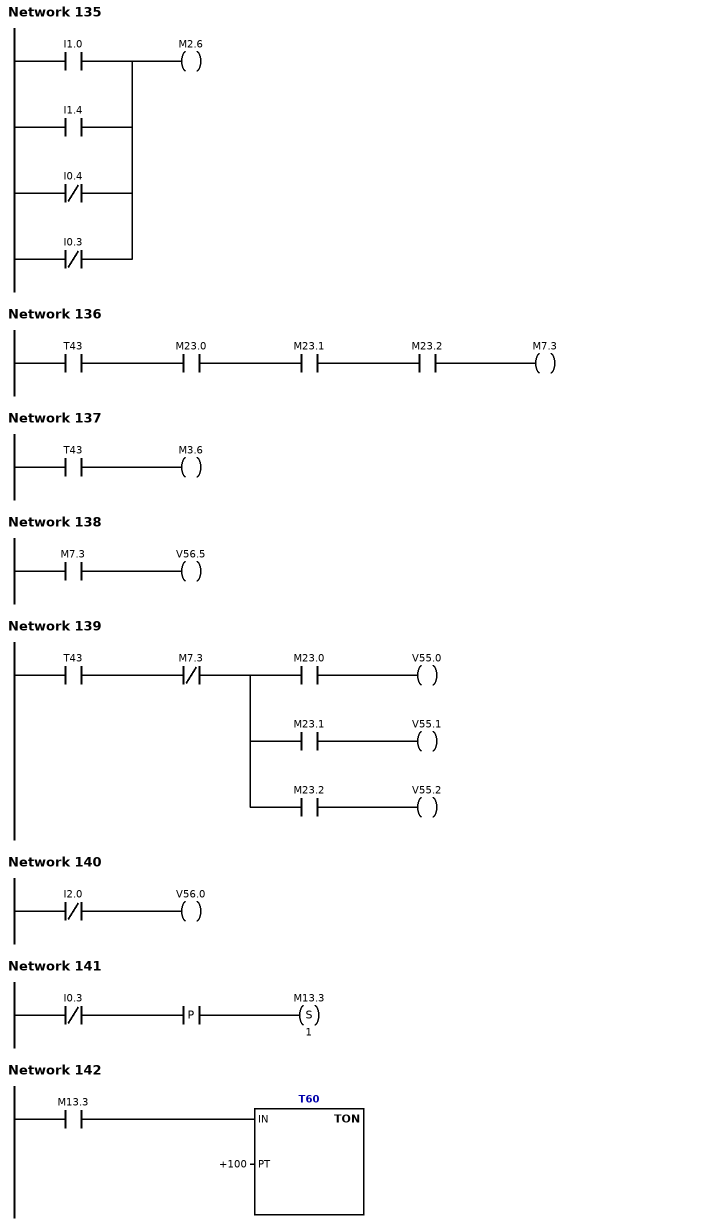
[picture p24: OB1 networks 135-142]
Network 135
LD     I1.0
O      I1.4
ON     I0.4
ON     I0.3
=      M2.6
Network 136
LD     T43
A      M23.0
A      M23.1
A      M23.2
=      M7.3
Network 137
LD     T43
=      M3.6
Network 138
LD     M7.3
=      V56.5
Network 139
LD     T43
AN     M7.3
LPS
A      M23.0
=      V55.0
LRD
A      M23.1
=      V55.1
LPP
A      M23.2
=      V55.2
Network 140
LDN    I2.0
=      V56.0
Network 141
LDN    I0.3
EU
S      M13.3, 1
Network 142
LD     M13.3
TON    T60, +100
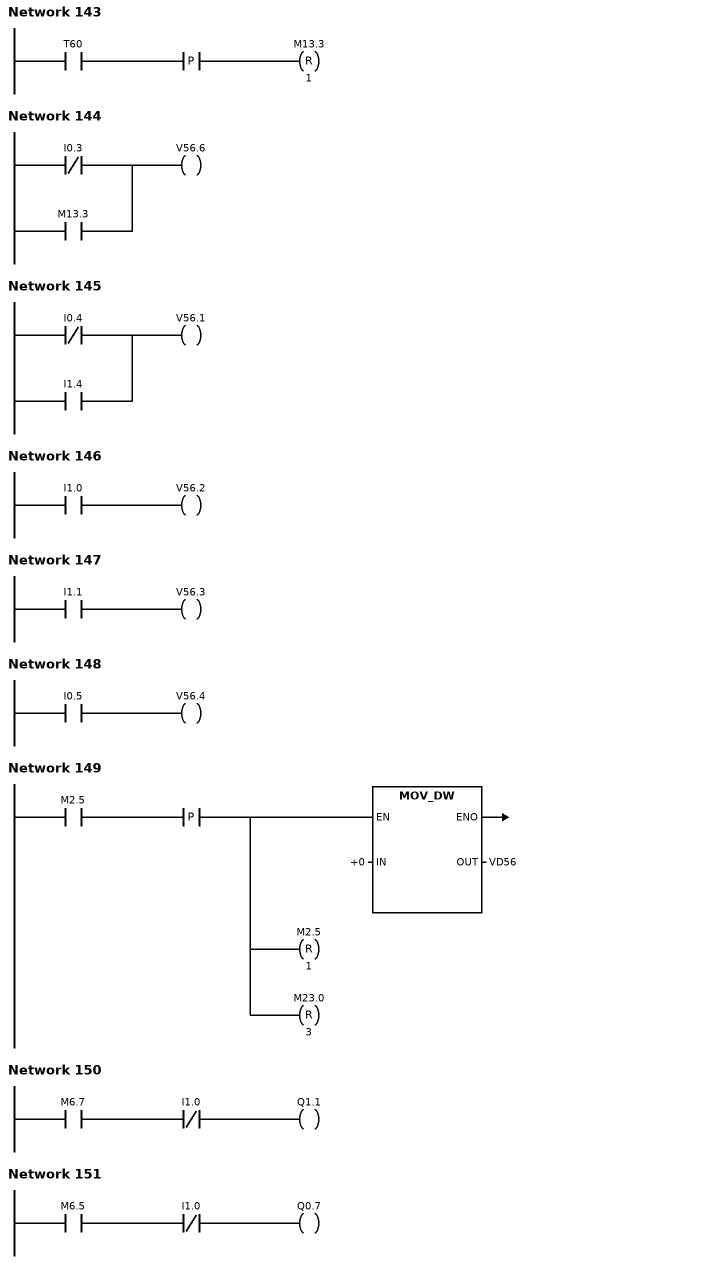
Network 143
LD     T60
EU
R      M13.3, 1
Network 144
LDN    I0.3
O      M13.3
=      V56.6
Network 145
LDN    I0.4
O      I1.4
=      V56.1
Network 146
LD     I1.0
=      V56.2
Network 147
LD     I1.1
=      V56.3
Network 148
LD     I0.5
=      V56.4
Network 149
LD     M2.5
EU
MOVD   +0, VD56
R      M2.5, 1
R      M23.0, 3
Network 150
LD     M6.7
AN     I1.0
=      Q1.1
Network 151
LD     M6.5
AN     I1.0
=      Q0.7
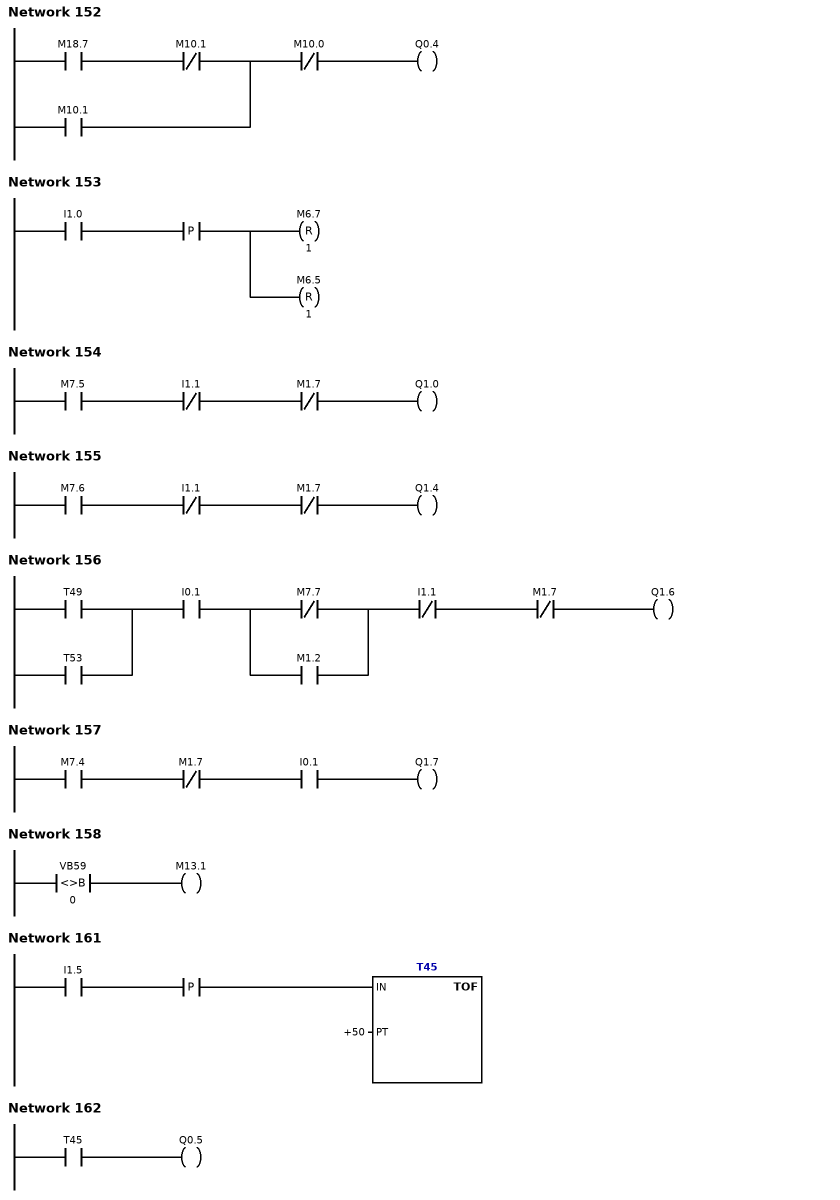
Network 152
LD     M18.7
AN     M10.1
O      M10.1
AN     M10.0
=      Q0.4
Network 153
LD     I1.0
EU
R      M6.7, 1
R      M6.5, 1
Network 154
LD     M7.5
AN     I1.1
AN     M1.7
=      Q1.0
Network 155
LD     M7.6
AN     I1.1
AN     M1.7
=      Q1.4
Network 156
LD     T49
O      T53
A      I0.1
LDN    M7.7
O      M1.2
ALD
AN     I1.1
AN     M1.7
=      Q1.6
Network 157
LD     M7.4
AN     M1.7
A      I0.1
=      Q1.7
Network 158
LDB<>  VB59, 0
=      M13.1
Network 161
LD     I1.5
EU
TOF    T45, +50
Network 162
LD     T45
=      Q0.5
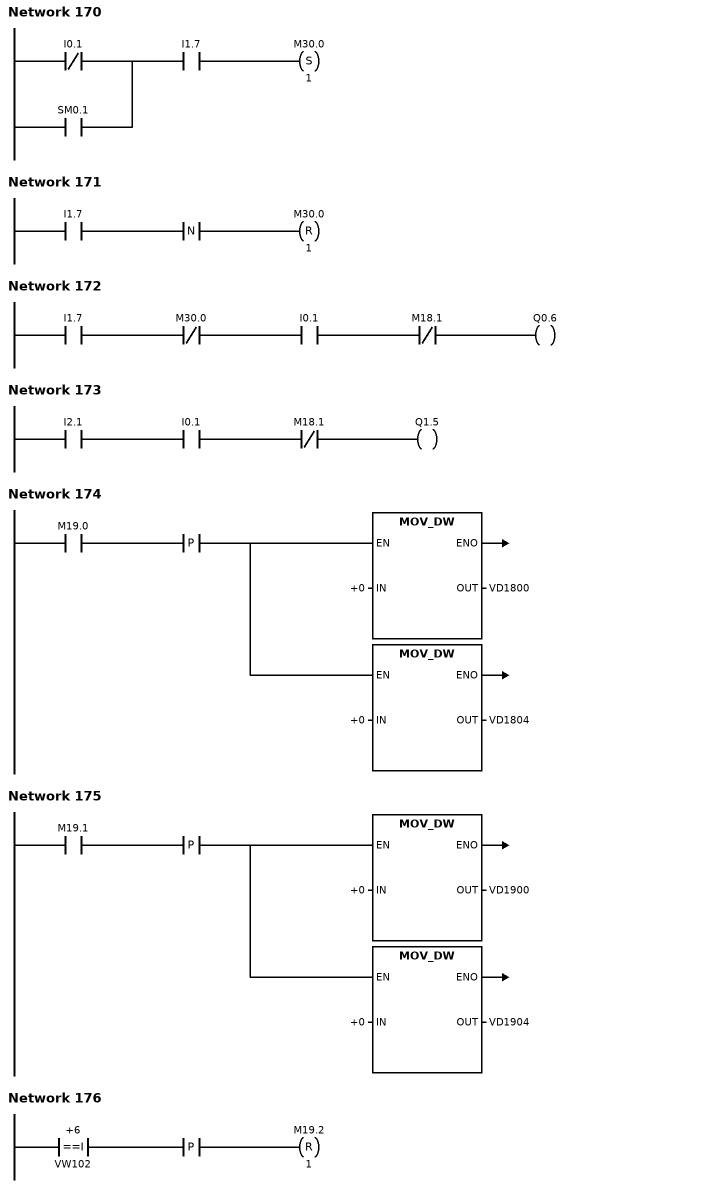
Network 170
LDN    I0.1
O      SM0.1
A      I1.7
S      M30.0, 1
Network 171
LD     I1.7
ED
R      M30.0, 1
Network 172
LD     I1.7
AN     M30.0
A      I0.1
AN     M18.1
=      Q0.6
Network 173
LD     I2.1
A      I0.1
AN     M18.1
=      Q1.5
Network 174
LD     M19.0
EU
MOVD   +0, VD1800
MOVD   +0, VD1804
Network 175
LD     M19.1
EU
MOVD   +0, VD1900
MOVD   +0, VD1904
Network 176
LDW=   +6, VW102
EU
R      M19.2, 1
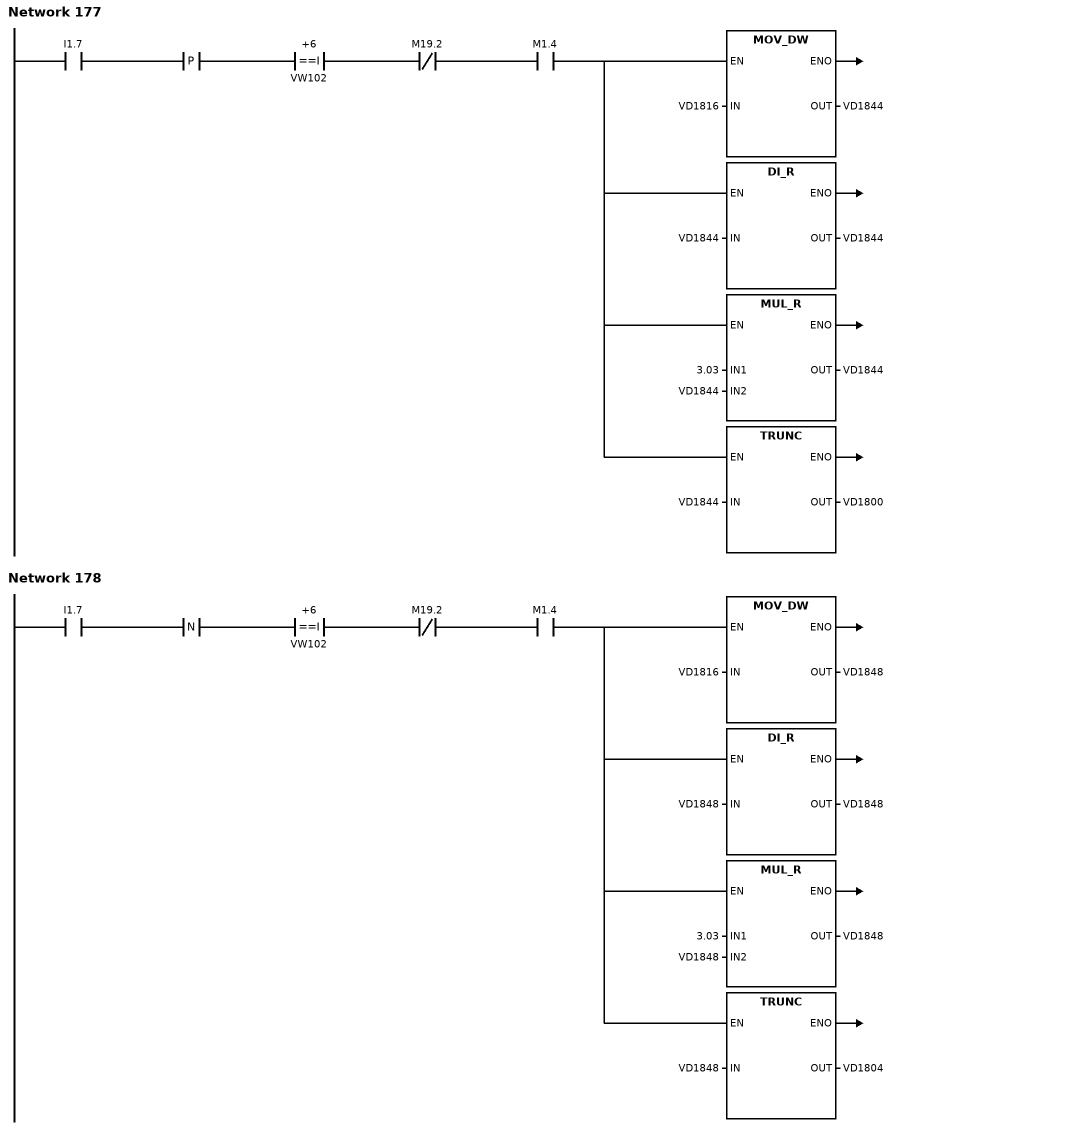
Network 177
LD     I1.7
EU
AW=    +6, VW102
AN     M19.2
A      M1.4
MOVD   VD1816, VD1844
DTR    VD1844, VD1844
*R     3.03, VD1844
TRUNC  VD1844, VD1800
Network 178
LD     I1.7
ED
AW=    +6, VW102
AN     M19.2
A      M1.4
MOVD   VD1816, VD1848
DTR    VD1848, VD1848
*R     3.03, VD1848
TRUNC  VD1848, VD1804
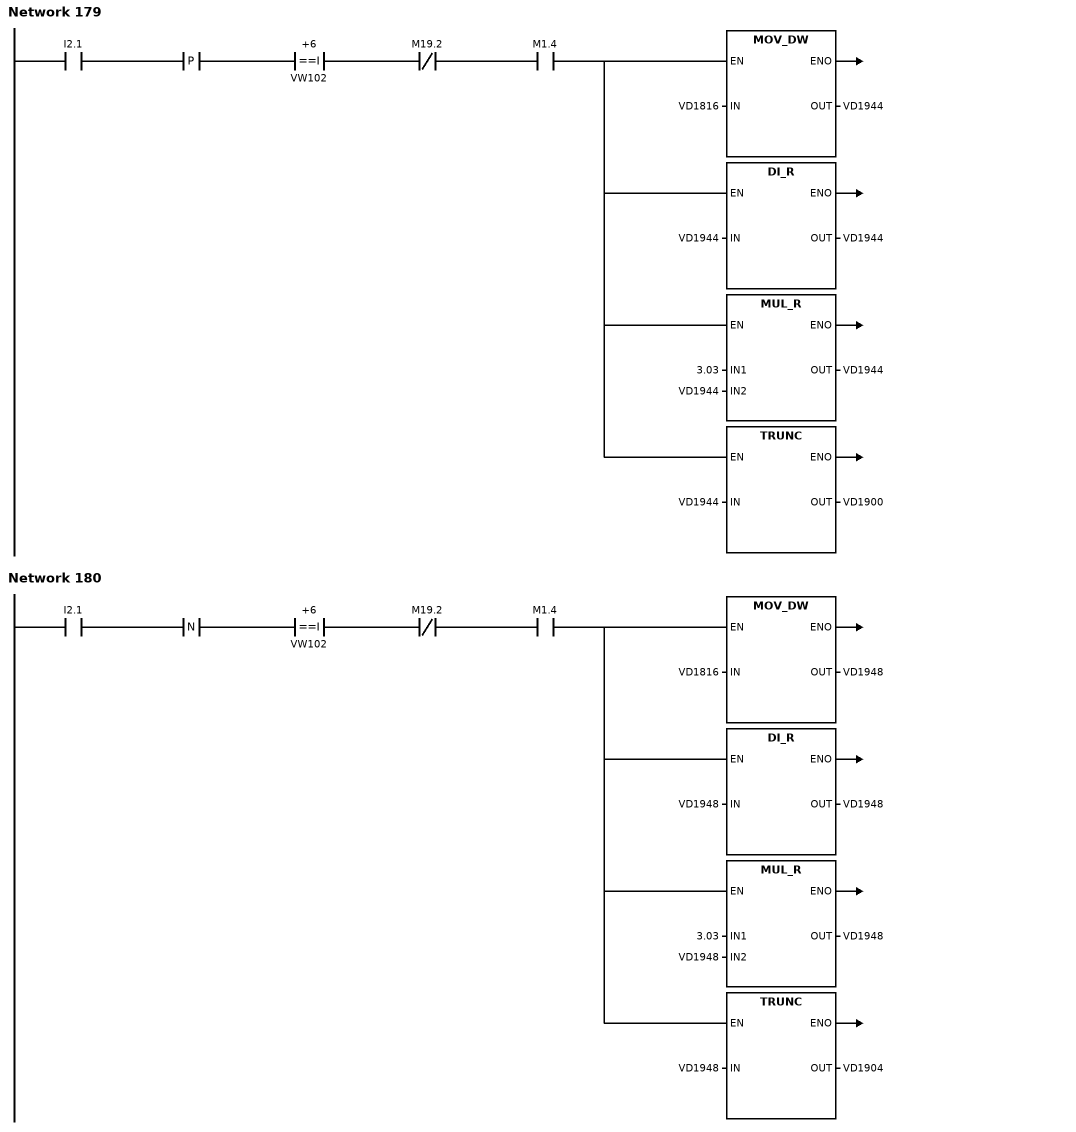
Network 179
LD     I2.1
EU
AW=    +6, VW102
AN     M19.2
A      M1.4
MOVD   VD1816, VD1944
DTR    VD1944, VD1944
*R     3.03, VD1944
TRUNC  VD1944, VD1900
Network 180
LD     I2.1
ED
AW=    +6, VW102
AN     M19.2
A      M1.4
MOVD   VD1816, VD1948
DTR    VD1948, VD1948
*R     3.03, VD1948
TRUNC  VD1948, VD1904
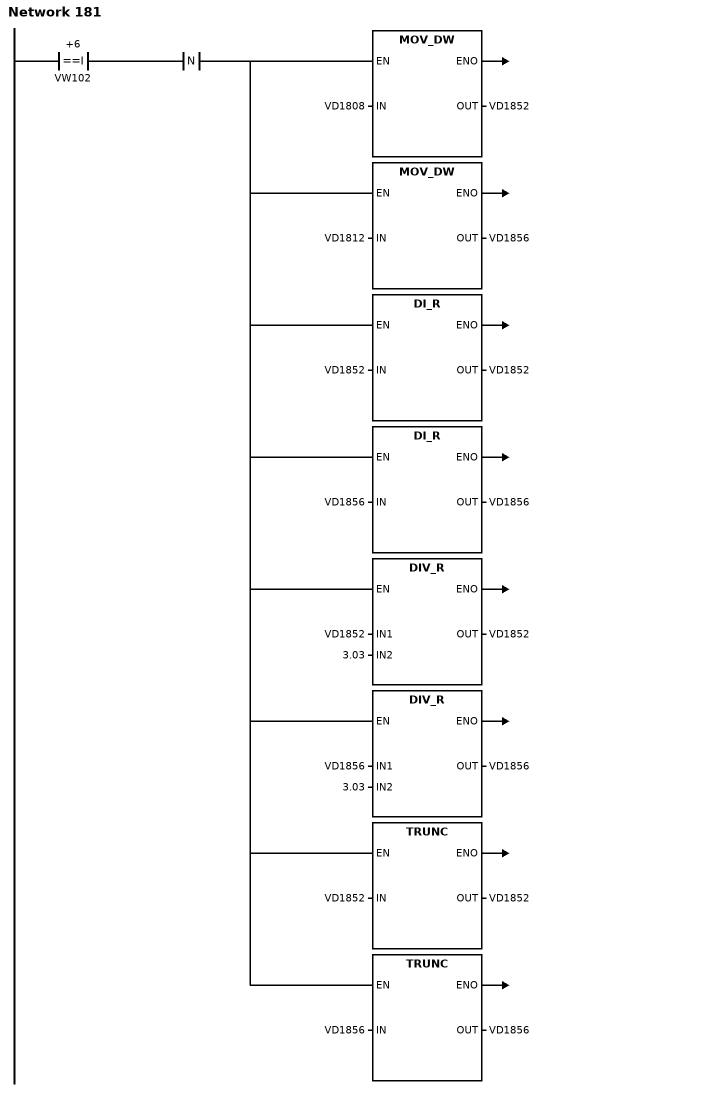
Network 181
LDW=   +6, VW102
ED
MOVD   VD1808, VD1852
MOVD   VD1812, VD1856
DTR    VD1852, VD1852
DTR    VD1856, VD1856
/R     3.03, VD1852
/R     3.03, VD1856
TRUNC  VD1852, VD1852
TRUNC  VD1856, VD1856
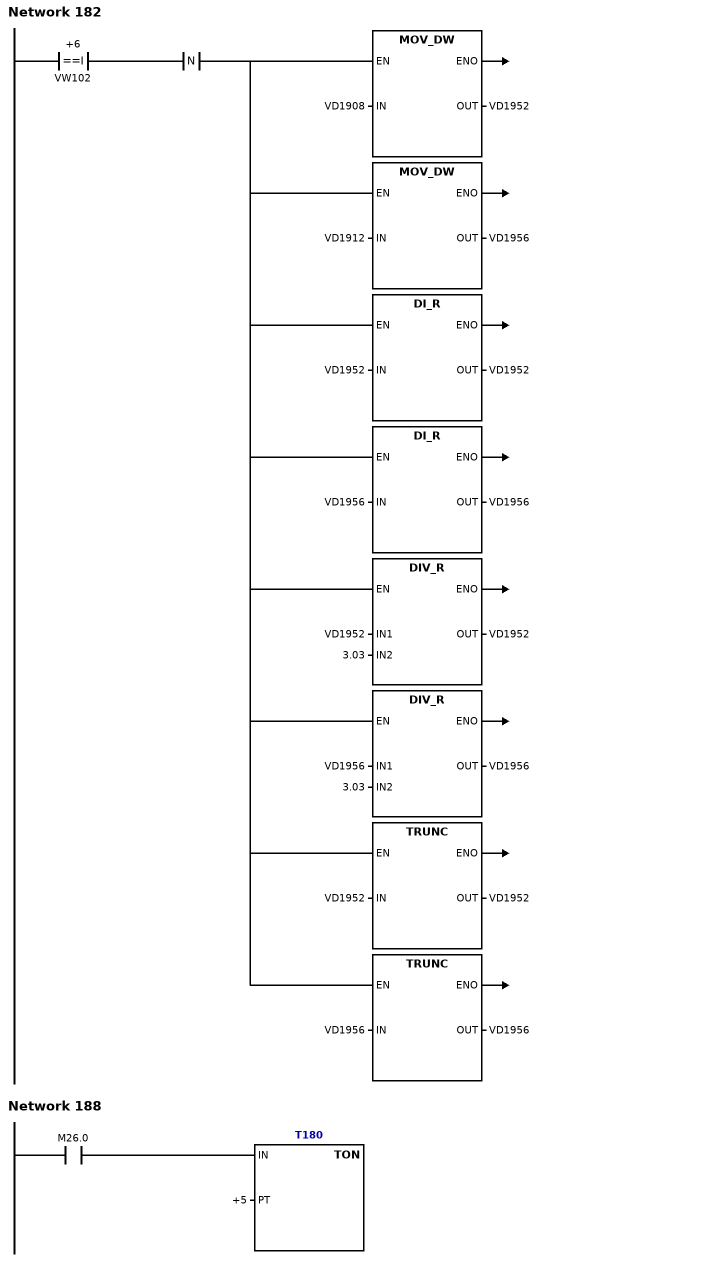
Network 182
LDW=   +6, VW102
ED
MOVD   VD1908, VD1952
MOVD   VD1912, VD1956
DTR    VD1952, VD1952
DTR    VD1956, VD1956
/R     3.03, VD1952
/R     3.03, VD1956
TRUNC  VD1952, VD1952
TRUNC  VD1956, VD1956
Network 188
LD     M26.0
TON    T180, +5
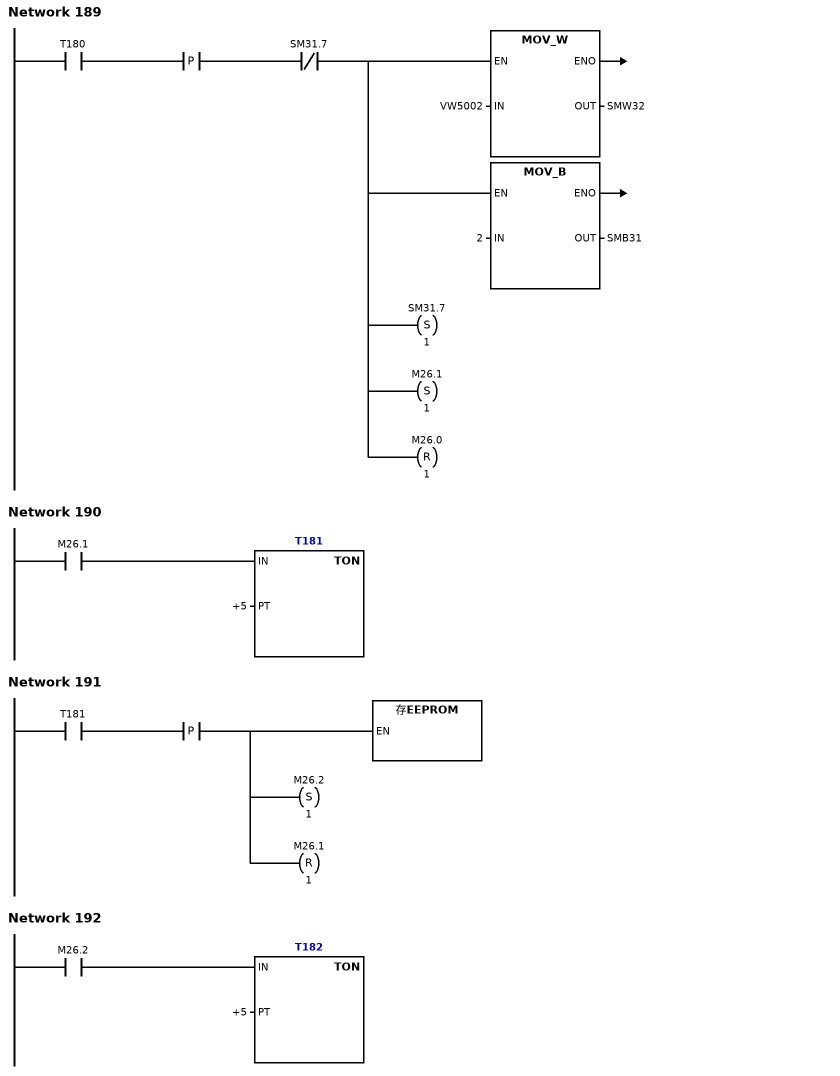
Network 189
LD     T180
EU
AN     SM31.7
MOVW   VW5002, SMW32
MOVB   2, SMB31
S      SM31.7, 1
S      M26.1, 1
R      M26.0, 1
Network 190
LD     M26.1
TON    T181, +5
Network 191
LD     T181
EU
CALL   存EEPROM:SBR7
S      M26.2, 1
R      M26.1, 1
Network 192
LD     M26.2
TON    T182, +5
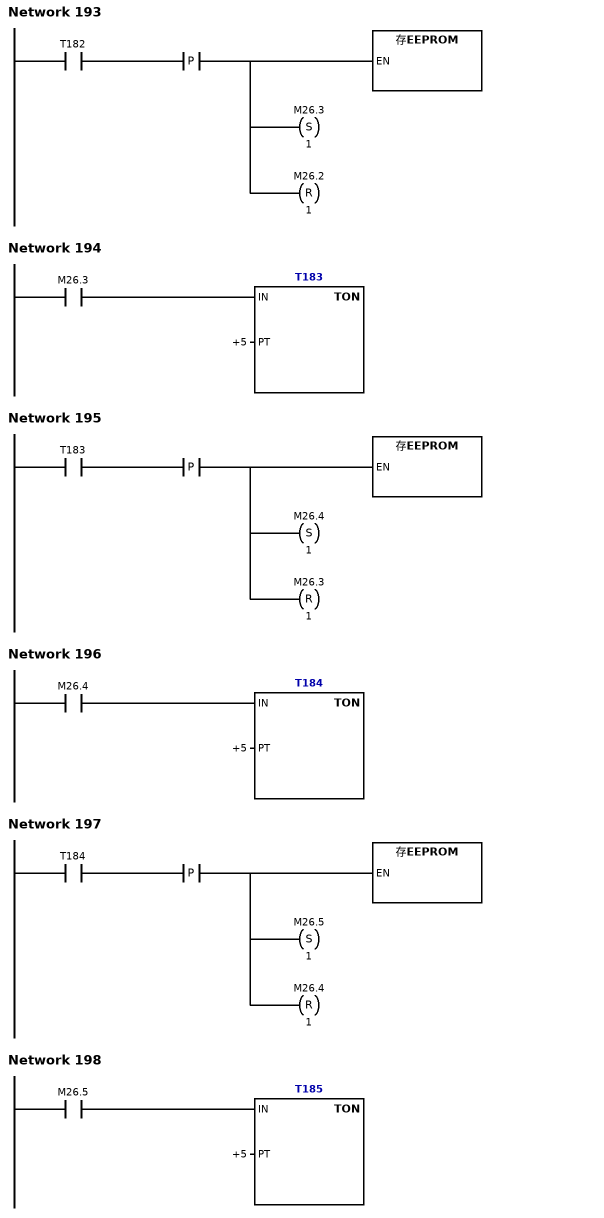
Network 193
LD     T182
EU
CALL   存EEPROM:SBR7
S      M26.3, 1
R      M26.2, 1
Network 194
LD     M26.3
TON    T183, +5
Network 195
LD     T183
EU
CALL   存EEPROM:SBR7
S      M26.4, 1
R      M26.3, 1
Network 196
LD     M26.4
TON    T184, +5
Network 197
LD     T184
EU
CALL   存EEPROM:SBR7
S      M26.5, 1
R      M26.4, 1
Network 198
LD     M26.5
TON    T185, +5
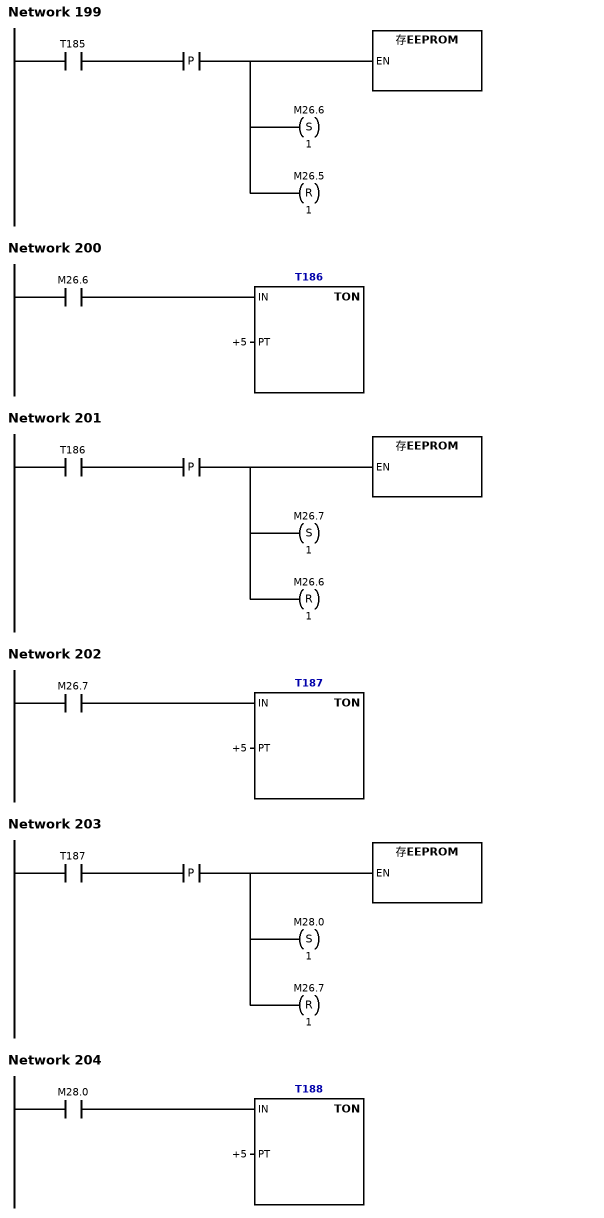
Network 199
LD     T185
EU
CALL   存EEPROM:SBR7
S      M26.6, 1
R      M26.5, 1
Network 200
LD     M26.6
TON    T186, +5
Network 201
LD     T186
EU
CALL   存EEPROM:SBR7
S      M26.7, 1
R      M26.6, 1
Network 202
LD     M26.7
TON    T187, +5
Network 203
LD     T187
EU
CALL   存EEPROM:SBR7
S      M28.0, 1
R      M26.7, 1
Network 204
LD     M28.0
TON    T188, +5
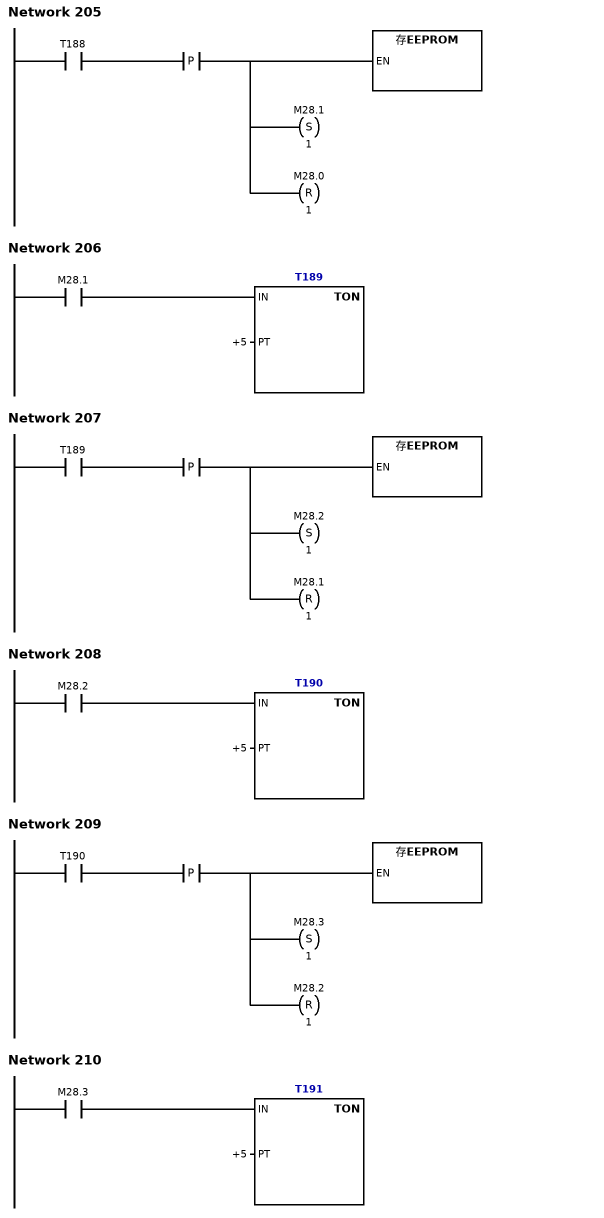
Network 205
LD     T188
EU
CALL   存EEPROM:SBR7
S      M28.1, 1
R      M28.0, 1
Network 206
LD     M28.1
TON    T189, +5
Network 207
LD     T189
EU
CALL   存EEPROM:SBR7
S      M28.2, 1
R      M28.1, 1
Network 208
LD     M28.2
TON    T190, +5
Network 209
LD     T190
EU
CALL   存EEPROM:SBR7
S      M28.3, 1
R      M28.2, 1
Network 210
LD     M28.3
TON    T191, +5
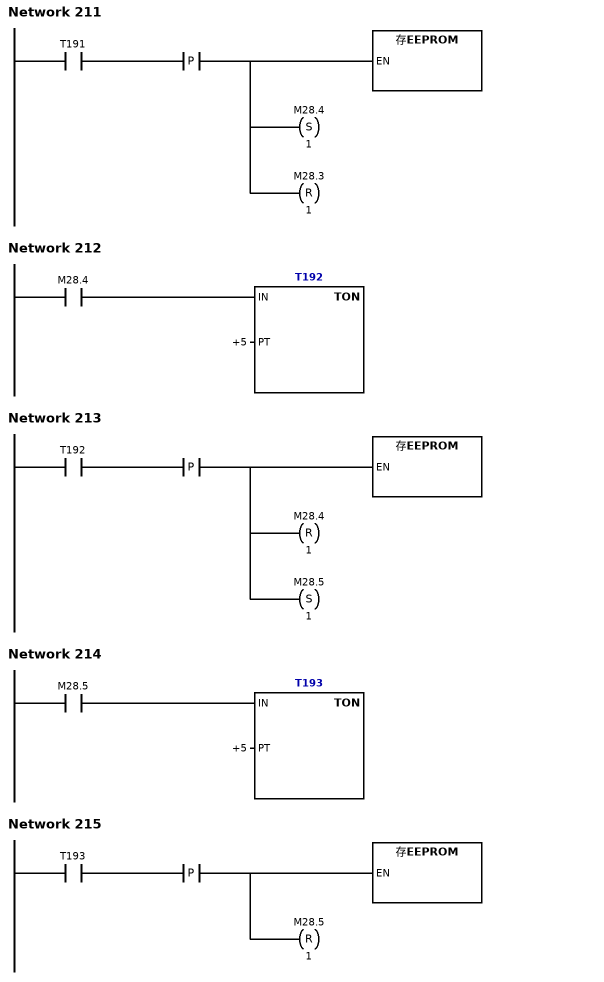
Network 211
LD     T191
EU
CALL   存EEPROM:SBR7
S      M28.4, 1
R      M28.3, 1
Network 212
LD     M28.4
TON    T192, +5
Network 213
LD     T192
EU
CALL   存EEPROM:SBR7
R      M28.4, 1
S      M28.5, 1
Network 214
LD     M28.5
TON    T193, +5
Network 215
LD     T193
EU
CALL   存EEPROM:SBR7
R      M28.5, 1
END_ORGANIZATION_BLOCK

SUBROUTINE_BLOCK 初始化:SBR0
TITLE=子程序注释
BEGIN
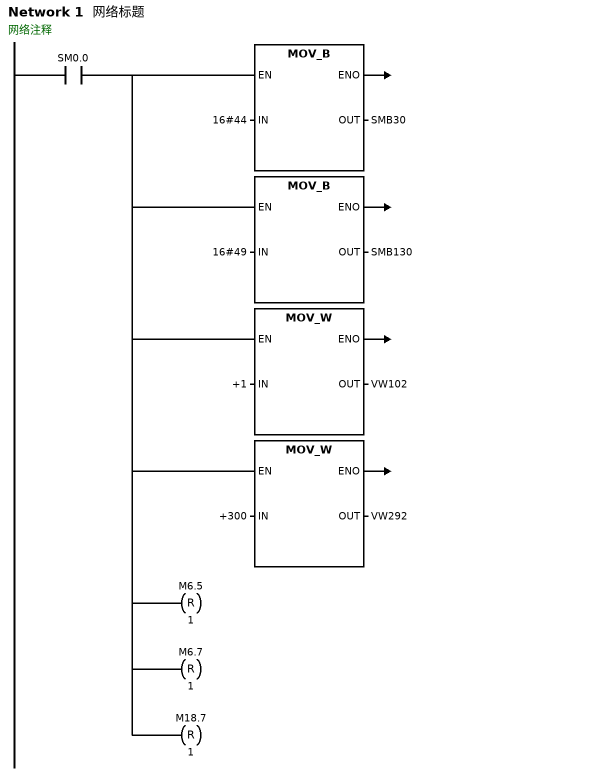
Network 1 // 网络标题
// 网络注释
LD     SM0.0
MOVB   16#44, SMB30
MOVB   16#49, SMB130
MOVW   +1, VW102
MOVW   +300, VW292
R      M6.5, 1
R      M6.7, 1
R      M18.7, 1
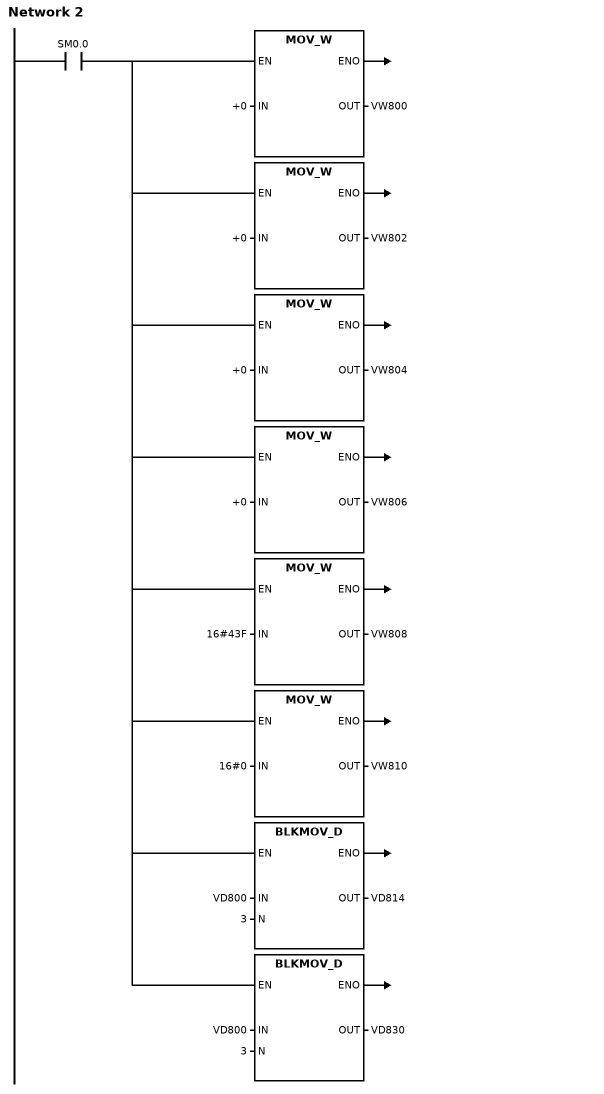
Network 2
LD     SM0.0
MOVW   +0, VW800
MOVW   +0, VW802
MOVW   +0, VW804
MOVW   +0, VW806
MOVW   16#43F, VW808
MOVW   16#0, VW810
BMD    VD800, VD814, 3
BMD    VD800, VD830, 3
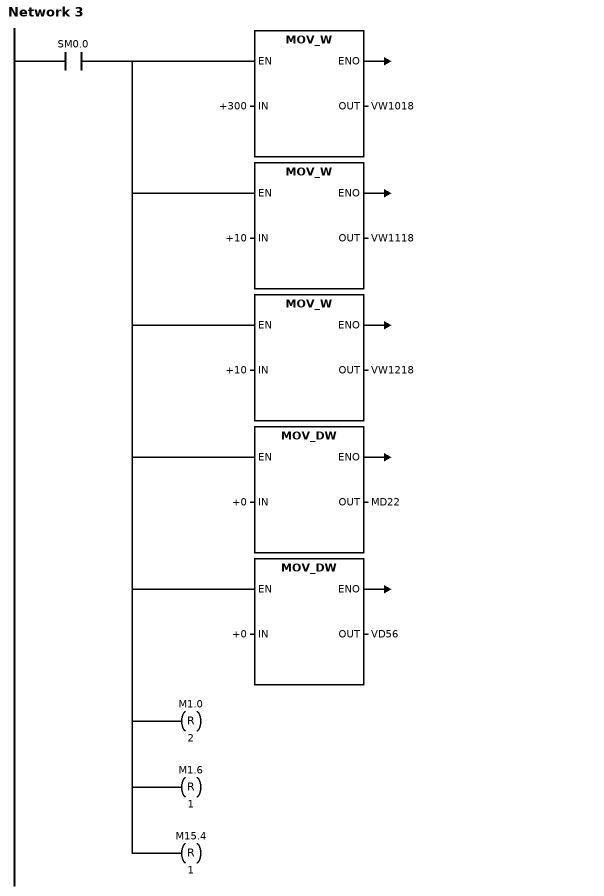
Network 3
LD     SM0.0
MOVW   +300, VW1018
MOVW   +10, VW1118
MOVW   +10, VW1218
MOVD   +0, MD22
MOVD   +0, VD56
R      M1.0, 2
R      M1.6, 1
R      M15.4, 1
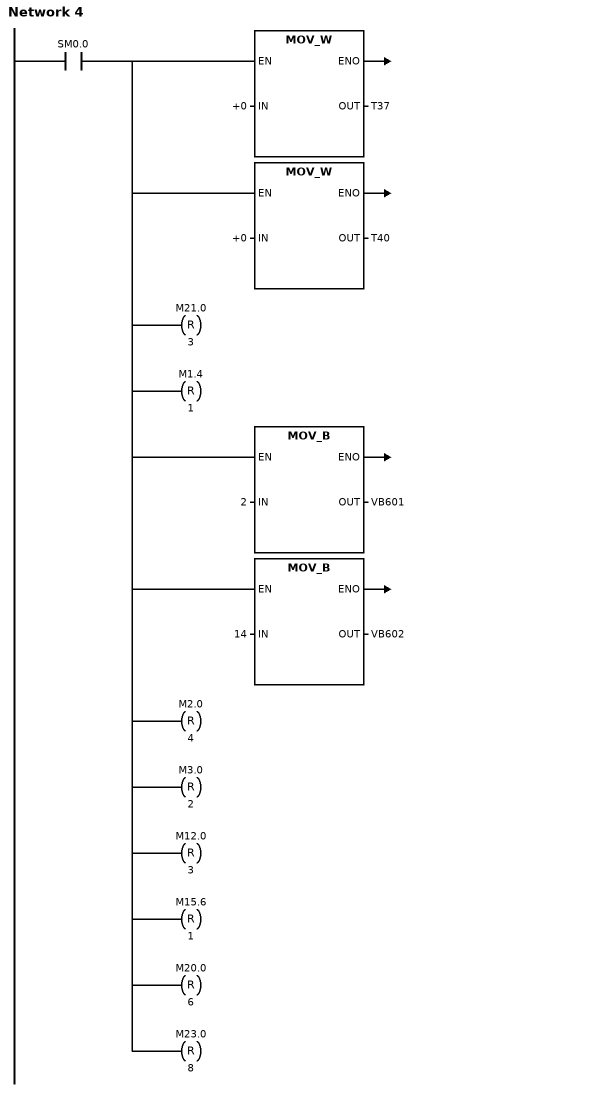
Network 4
LD     SM0.0
MOVW   +0, T37
MOVW   +0, T40
R      M21.0, 3
R      M1.4, 1
MOVB   2, VB601
MOVB   14, VB602
R      M2.0, 4
R      M3.0, 2
R      M12.0, 3
R      M15.6, 1
R      M20.0, 6
R      M23.0, 8
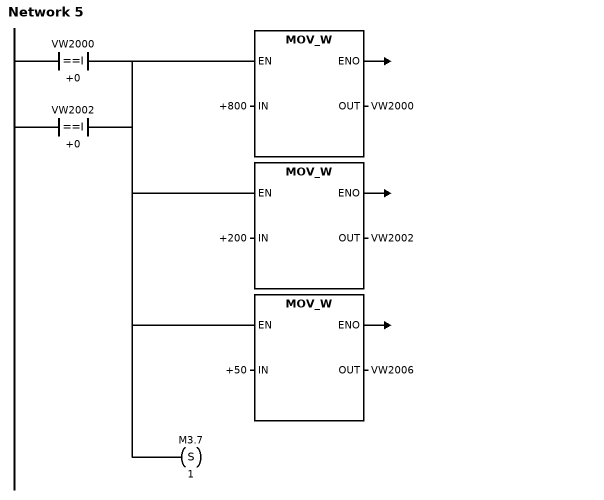
Network 5
LDW=   VW2000, +0
OW=    VW2002, +0
MOVW   +800, VW2000
MOVW   +200, VW2002
MOVW   +50, VW2006
S      M3.7, 1
END_SUBROUTINE_BLOCK

SUBROUTINE_BLOCK 发送命令:SBR1
TITLE=
BEGIN
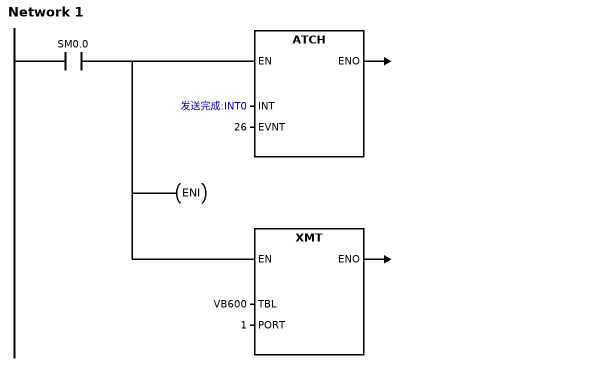
Network 1
LD     SM0.0
ATCH   发送完成:INT0, 26
ENI
XMT    VB600, 1
END_SUBROUTINE_BLOCK

SUBROUTINE_BLOCK 生成BCC:SBR2
TITLE=
BEGIN
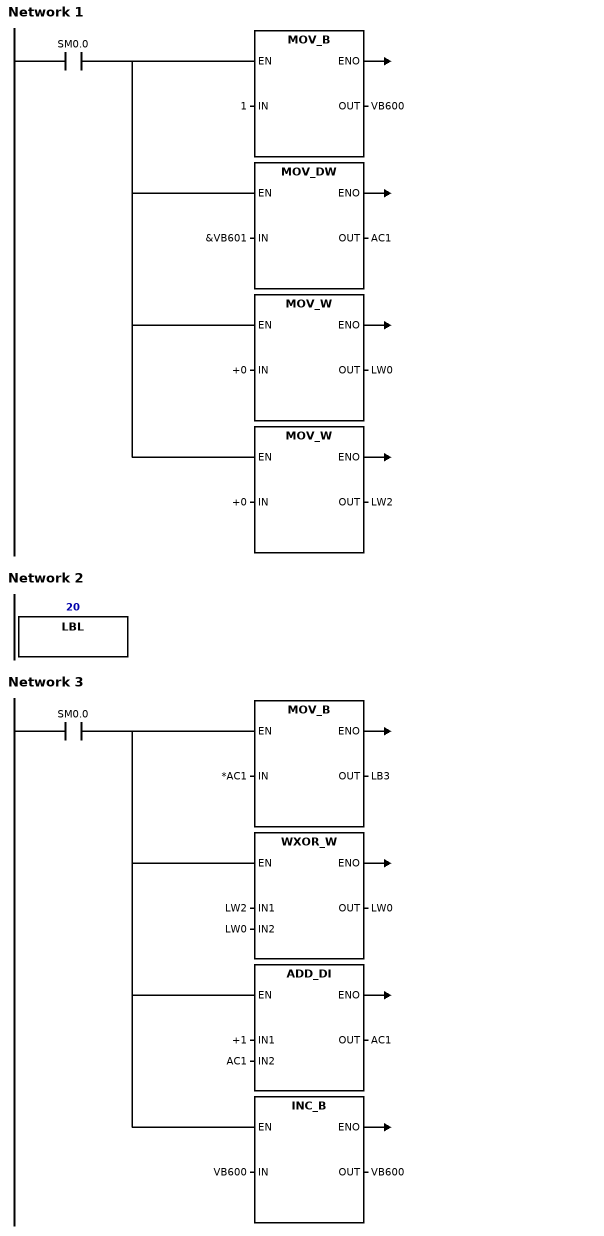
Network 1
LD     SM0.0
MOVB   1, VB600
MOVD   &VB601, AC1
MOVW   +0, LW0
MOVW   +0, LW2
Network 2
LBL    20
Network 3
LD     SM0.0
MOVB   *AC1, LB3
XORW   LW2, LW0
+D     +1, AC1
INCB   VB600
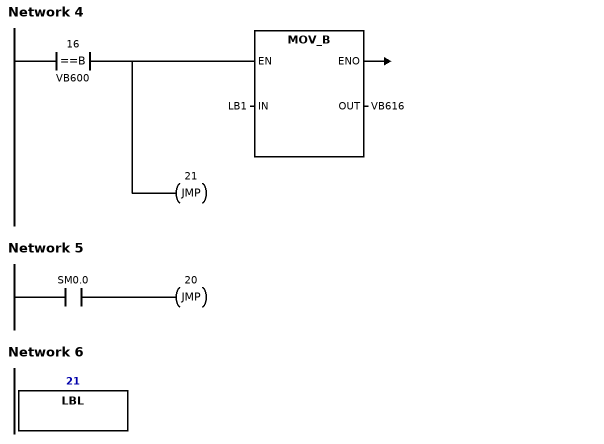
Network 4
LDB=   16, VB600
MOVB   LB1, VB616
JMP    21
Network 5
LD     SM0.0
JMP    20
Network 6
LBL    21
END_SUBROUTINE_BLOCK

SUBROUTINE_BLOCK 变频器读_写检查:SBR3
TITLE=
BEGIN
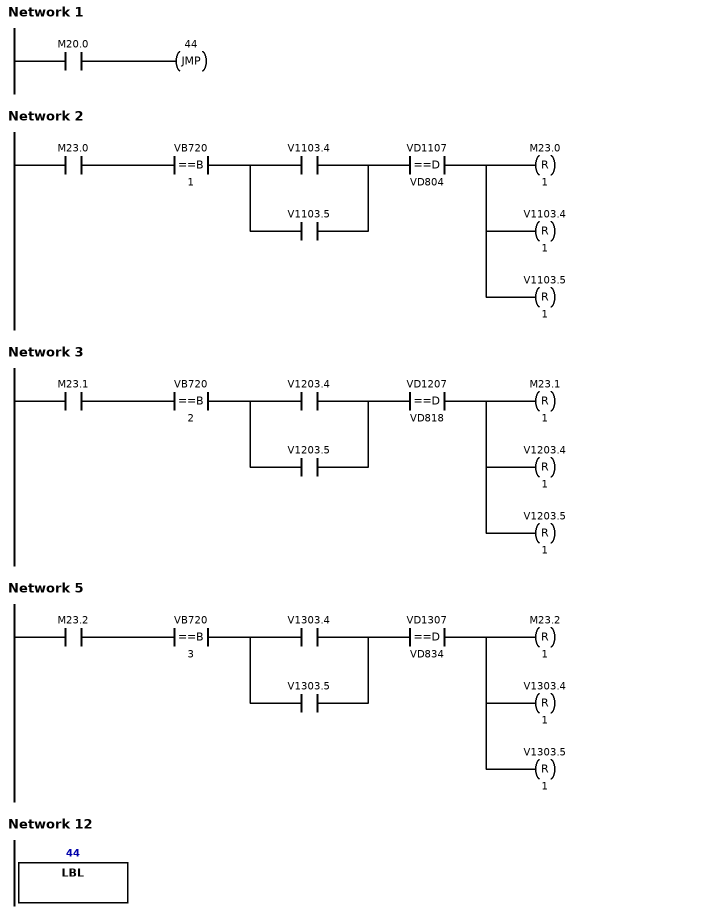
Network 1
LD     M20.0
JMP    44
Network 2
LD     M23.0
AB=    VB720, 1
LD     V1103.4
O      V1103.5
ALD
AD=    VD1107, VD804
R      M23.0, 1
R      V1103.4, 1
R      V1103.5, 1
Network 3
LD     M23.1
AB=    VB720, 2
LD     V1203.4
O      V1203.5
ALD
AD=    VD1207, VD818
R      M23.1, 1
R      V1203.4, 1
R      V1203.5, 1
Network 5
LD     M23.2
AB=    VB720, 3
LD     V1303.4
O      V1303.5
ALD
AD=    VD1307, VD834
R      M23.2, 1
R      V1303.4, 1
R      V1303.5, 1
Network 12
LBL    44
END_SUBROUTINE_BLOCK

SUBROUTINE_BLOCK 启停命令控制:SBR4
TITLE=
BEGIN
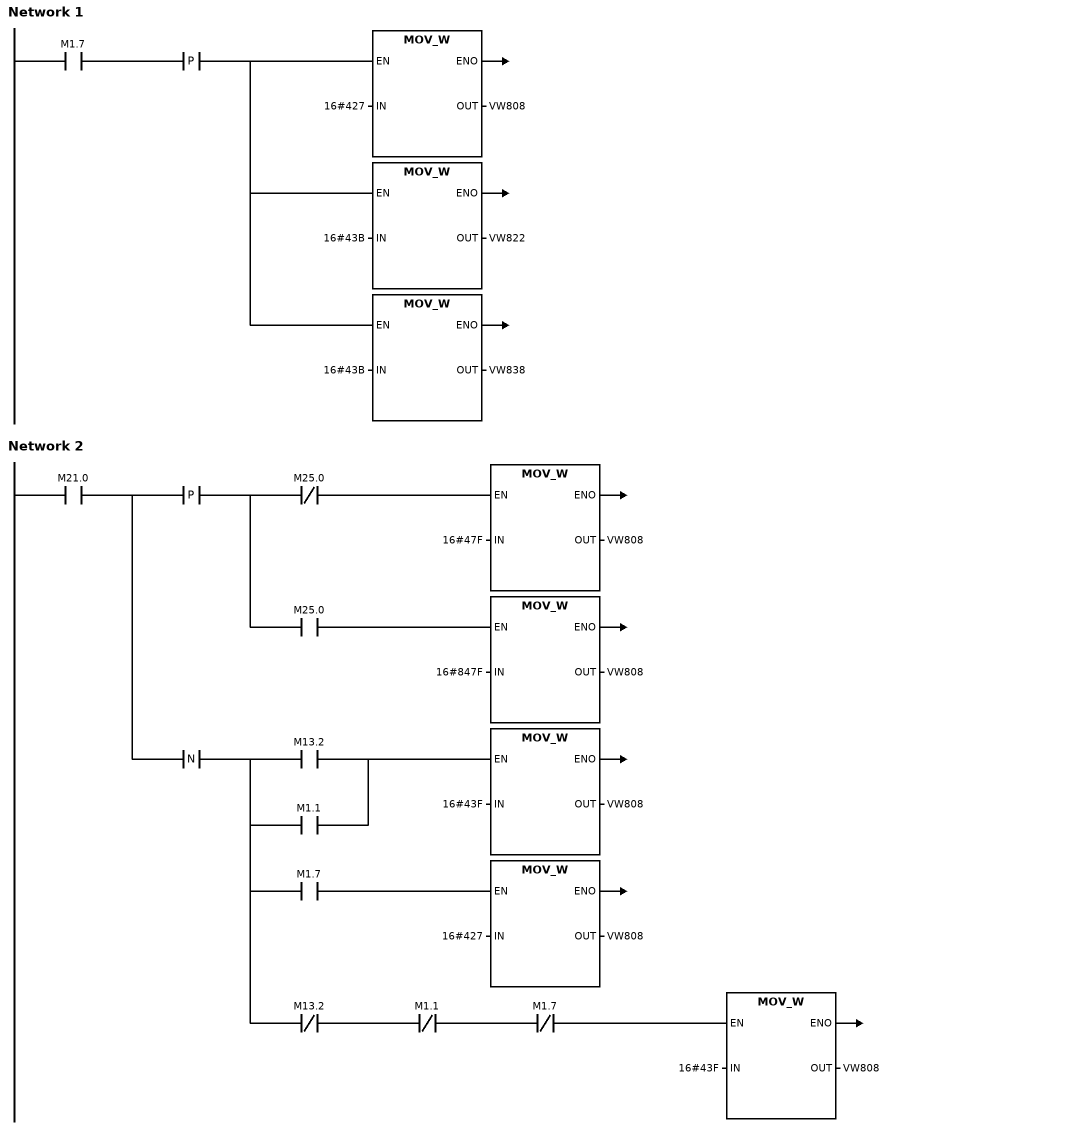
Network 1
LD     M1.7
EU
MOVW   16#427, VW808
MOVW   16#43B, VW822
MOVW   16#43B, VW838
Network 2
LD     M21.0
LPS
EU
LPS
AN     M25.0
MOVW   16#47F, VW808
LPP
A      M25.0
MOVW   16#847F, VW808
LPP
ED
LPS
LD     M13.2
O      M1.1
ALD
MOVW   16#43F, VW808
LPP
LPS
A      M1.7
MOVW   16#427, VW808
LPP
AN     M13.2
AN     M1.1
AN     M1.7
MOVW   16#43F, VW808
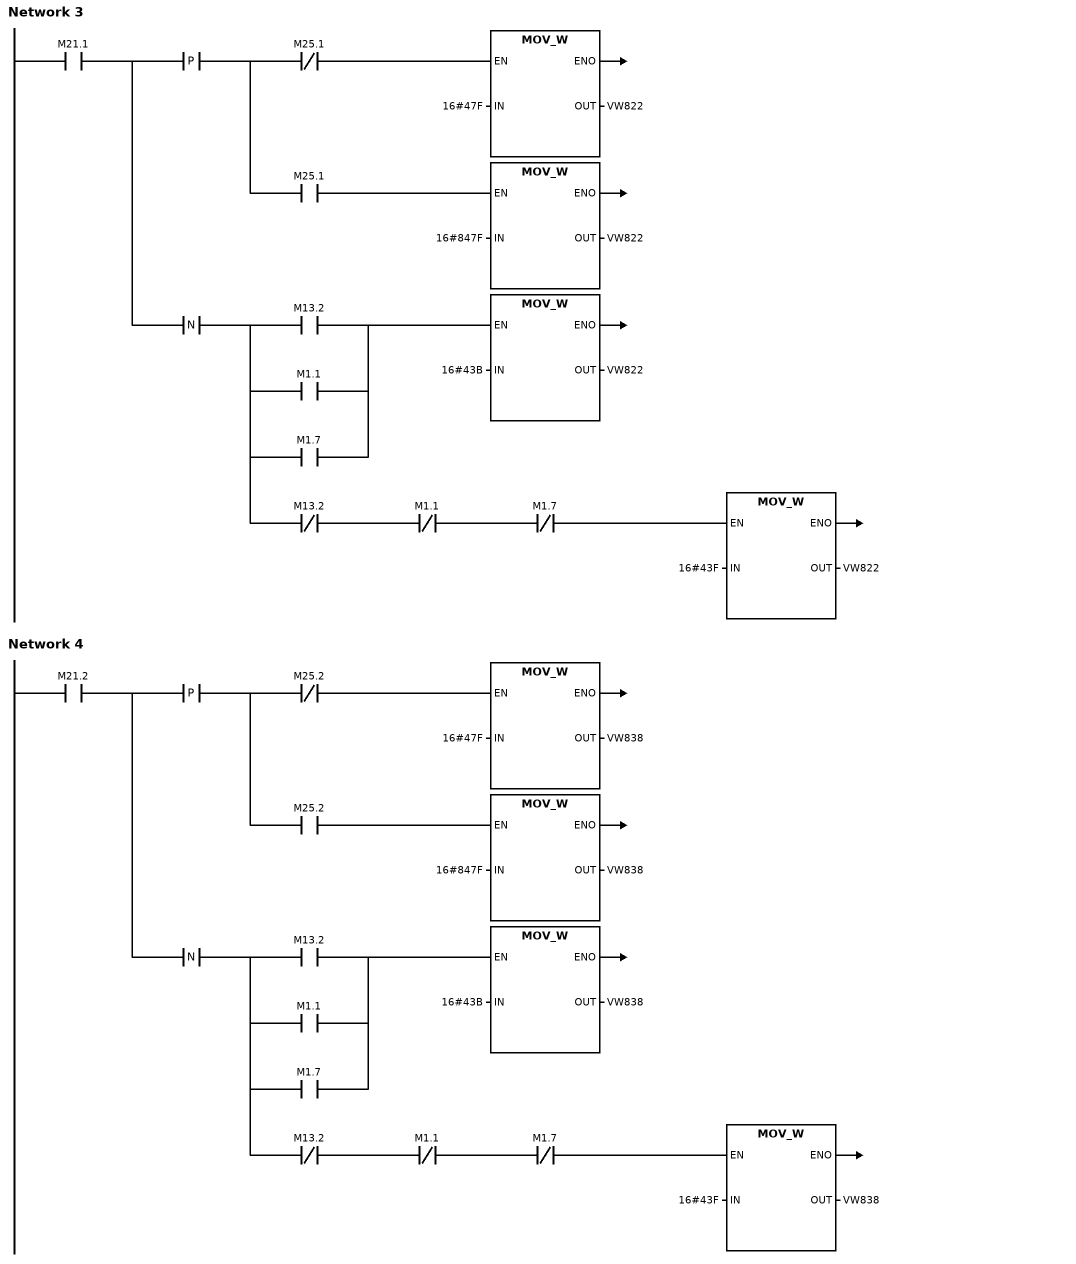
Network 3
LD     M21.1
LPS
EU
LPS
AN     M25.1
MOVW   16#47F, VW822
LPP
A      M25.1
MOVW   16#847F, VW822
LPP
ED
LPS
LD     M13.2
O      M1.1
O      M1.7
ALD
MOVW   16#43B, VW822
LPP
AN     M13.2
AN     M1.1
AN     M1.7
MOVW   16#43F, VW822
Network 4
LD     M21.2
LPS
EU
LPS
AN     M25.2
MOVW   16#47F, VW838
LPP
A      M25.2
MOVW   16#847F, VW838
LPP
ED
LPS
LD     M13.2
O      M1.1
O      M1.7
ALD
MOVW   16#43B, VW838
LPP
AN     M13.2
AN     M1.1
AN     M1.7
MOVW   16#43F, VW838
END_SUBROUTINE_BLOCK

SUBROUTINE_BLOCK 存工艺:SBR5
TITLE=
BEGIN
